// TwinCAT 3 PLC project PLC
// ProgramVersion: 3.1.4024.0
// libraries:
//   Tc2_Standard, * (Beckhoff Automation GmbH)
//   Tc2_System, * (Beckhoff Automation GmbH)
//   Tc3_EventLogger, * (Beckhoff Automation GmbH)
//   Tc3_Module, * (Beckhoff Automation GmbH)
// project tree:
//   GVLs/ GVL.TcGVL
//   / PlcTask.TcTTO
//   POUs/ FB_ALARM.TcPOU, FB_ListenerTest.TcPOU, FB_SampleListener.TcPOU, TYP_ALARM_INTERFACE.TcDUT, MAIN.TcPOU
// real-time tasks:
//   TASK PlcTask: cycle T#10ms, priority 20, ADS port 350

CONFIGURATION PLC
    RESOURCE PLC ON TwinCAT3
        TASK PlcTask(INTERVAL := T#10ms, PRIORITY := 20);
        PROGRAM MAIN WITH PlcTask : MAIN;
    END_RESOURCE
END_CONFIGURATION

// ---- POUs/TYP_ALARM_INTERFACE.TcDUT
TYPE TYP_ALARM_INTERFACE :
STRUCT
	bActivate : BOOL;
	bConfirm : BOOL;
	sMessage : STRING;
	sSourceMessage : STRING;
	nEventID : UDINT;
	nSourceID : UDINT;
END_STRUCT
END_TYPE

// ---- GVLs/GVL.TcGVL
{attribute 'qualified_only'}
VAR_GLOBAL
	{attribute 'OPC.UA.DA' := '1'}
	{attribute 'OPC.UA.DA.StructuredType' := '1'}
	arrAlarms : ARRAY[0..99] OF TYP_ALARMS;
END_VAR

// ---- POUs/MAIN.TcPOU
PROGRAM MAIN
VAR
	GeneralAlarms : ARRAY[0..2] OF TYP_ALARM_INTERFACE :=
	[(nEventID:=3, nSourceID:=101, sMessage:='MESSAGE 1', sSourceMessage:='SOURCE 1'),
	(nEventID:=3, nSourceID:=202, sMessage:='MESSAGE 2', sSourceMessage:='SOURCE 2'),
	(nEventID:=3, nSourceID:=303, sMessage:='MESSAGE 3', sSourceMessage:='SOURCE 3')];
	
	fbGeneralAlarms : ARRAY [0..2] OF FB_ALARM;
	fbListener : FB_ListenerTest;
	bResetArray : BOOL;
	i: INT;
END_VAR

fbListener(arrAlarms:=GVL.arrAlarms);

FOR i:=0 TO 2 BY 1 DO
	fbGeneralAlarms[i](eventEntry:=TC_EVENTS.AlarmEventClass.General_alarm, 
			bEvt := GeneralAlarms[i].bActivate, 
			bConfirm := GeneralAlarms[i].bConfirm,
			sMessage := GeneralAlarms[i].sMessage,
			nUserEventID := GeneralAlarms[i].nEventID,
			nUserSourceID := GeneralAlarms[i].nSourceID,
			sSourceMessage := GeneralAlarms[i].sSourceMessage,
			arrAlarms := GVL.arrAlarms);
END_FOR	
		
IF bResetArray THEN
	memset(ADR(GVL.arrAlarms),0,SIZEOF(GVL.arrAlarms));
	bResetArray := FALSE;
END_IF

END_PROGRAM

// ---- POUs/FB_ALARM.TcPOU
FUNCTION_BLOCK FB_ALARM EXTENDS FB_TcAlarm
VAR_INPUT
	eventEntry : TcEventEntry;
	bEvt : BOOL;
	bConfirm : BOOL;
	nUserEventID : UDINT;
	nUserSourceID : UDINT;
	sMessage : STRING;
	sSourceMessage : STRING;
END_VAR
VAR_IN_OUT
	arrAlarms : ARRAY[*] OF TYP_ALARMS;
END_VAR
VAR_OUTPUT
END_VAR
VAR
	bInit : BOOL := TRUE;
	bMem : BOOL;
	fbMsg : FB_TcMessage;
	fbSourceInformation : FB_TcSourceInfo;
END_VAR

//INITIALISING THE ALARM WHEN THE RAISING OF THE ALARM IS REQUESTED
IF bEvt AND NOT bMem (*AND SUPER^.eConfirmationState <> TcEventConfirmationState.WaitForConfirmation*) THEN
	IF bInit THEN
		fbSourceInformation.Clear();
		fbSourceInformation.sName := sSourceMessage;
		fbSourceInformation.nId := nUserSourceID;
		eventEntry.nEventId := nUserEventID;
		SUPER^.CreateEx(eventEntry, TRUE, ipSourceInfo := fbSourceInformation);
		SUPER^.ipArguments.Clear().AddString(sMessage);
		bInit := FALSE;
	END_IF
END_IF

//AFTER INITIALISING, RAISE THE ALARM
IF NOT bInit THEN
	SUPER^.Raise(0);
	bInit := TRUE;
END_IF

//CLEARING THE ALARM
IF bMem AND NOT bEvt THEN
	SUPER^.Clear(0, FALSE);	
END_IF

//CONFIRMING THE ALARM
IF bConfirm THEN
	SUPER^.Confirm(0);
END_IF

bMem := bEvt;

END_FUNCTION_BLOCK

// ---- POUs/FB_ListenerTest.TcPOU
FUNCTION_BLOCK FB_ListenerTest
VAR_INPUT
END_VAR
VAR_IN_OUT
	arrAlarms : ARRAY[*] OF TYP_ALARMS;
END_VAR
VAR_OUTPUT
END_VAR
VAR
	hr : HRESULT;
	
	bSubscribe : BOOL := TRUE;
	bSubscribed : BOOL;
	bUnSubscribe : BOOL;
	
	fbListenerFilter : FB_TcEventFilter; 
	fbMessageListener : FB_SampleListener;
	
END_VAR

fbMessageListener.arrAlarms := arrAlarms;
fbMessageListener.Execute(); // retrieve messages and its texts

IF bSubscribe THEN 
	bSubscribe := FALSE;
	fbListenerFilter.Clear().EventClass.EqualTo(TC_EVENTS.AlarmEventClass.General_alarm.uuidEventClass); //define all events (messages and alarms) from this eventclass   
	hr := fbMessageListener.Subscribe2(fbListenerFilter); //subscribe to retrieve defined events
	IF SUCCEEDED(hr) THEN	
		bSubscribed := TRUE;
	END_IF
END_IF 

IF bUnSubscribe THEN 
	bUnSubscribe := FALSE;
	hr := fbMessageListener.Unsubscribe();
	IF SUCCEEDED(hr) THEN	
		bSubscribed := FALSE;
	END_IF
END_IF

END_FUNCTION_BLOCK

// ---- POUs/FB_SampleListener.TcPOU
FUNCTION_BLOCK FB_SampleListener EXTENDS FB_ListenerBase2
VAR_INPUT
END_VAR
VAR_IN_OUT
	arrAlarms : ARRAY[*] OF TYP_ALARMS;
END_VAR
VAR_OUTPUT
END_VAR
VAR
	sJsonAttribute : STRING (10000);	
	hr : HRESULT;
	
	nCntMessagesSent : INT;
	nCntAlarmsRaised : INT;
	nCntAlarmsConfirmed : INT;
	nCntAlarmsCleared : INT;
	
	//text retrieval of message
	fbRequestEventText : FB_RequestEventText;
	{attribute 'TcEncoding':='UTF-8'}
	sLastMessageText : STRING;
	bReqText : BOOL;
END_VAR

METHOD Execute : HRESULT
VAR_INPUT
END_VAR
Execute := SUPER^.Execute(); //retrieve events

//retrieve the text of a message
IF 	bReqText AND fbRequestEventText.bError THEN 
	sLastMessageText := 'Error';
	bReqText := FALSE; 
ELSIF bReqText AND NOT  fbRequestEventText.bBusy THEN
	fbRequestEventText.GetString(sLastMessageText, SIZEOF(sLastMessageText));
	bReqText := FALSE;
END_IF
END_METHOD

METHOD OnAlarmCleared : HRESULT
VAR_INPUT
	fbEvent : REFERENCE TO FB_TcEvent;
END_VAR
VAR
	i : INT;
	j : INT;
END_VAR
nCntAlarmsCleared := nCntAlarmsCleared + 1;

FOR i:=0 TO 99 BY 1 DO
	//CYCLING THRU THE ARRAY TO FIND IF A MATCHING ALARM EXISTS
	IF arrAlarms[i].AlarmID = fbEvent.nEventId AND arrAlarms[i].SourceID = fbEvent.ipSourceInfo.nId THEN
		//UPDATING THE CONFIRMED STATE
		arrAlarms[i].isActive := FALSE;	
	END_IF	 
	//IF ALARM IS (CONFIRMED AND NOT ACTIVE) THEN REMOVING THE ALARM FROM THE ARRAY
	IF arrAlarms[i].isConfirmed AND NOT arrAlarms[i].isActive THEN
		FOR j:=i TO 99 BY 1 DO
			arrAlarms[j]:=arrAlarms[j+1];
		END_FOR
	END_IF	
END_FOR

OnAlarmCleared := S_OK; // in order to receive more callbacks (Set <> S_OK in order to cancel the callbacks for this program cycle.)
END_METHOD

METHOD OnAlarmConfirmed : HRESULT
VAR_INPUT
	fbEvent : REFERENCE TO FB_TcEvent;
END_VAR
VAR
	i : INT;
	j: INT;
END_VAR
nCntAlarmsConfirmed := nCntAlarmsConfirmed + 1;

FOR i:=0 TO 99 BY 1 DO
	//CYCLING THRU THE ARRAY TO FIND IF A MATCHING ALARM EXISTS
	IF arrAlarms[i].AlarmID = fbEvent.nEventId AND arrAlarms[i].SourceID = fbEvent.ipSourceInfo.nId THEN
		//UPDATING THE CONFIRMED STATE
		arrAlarms[i].isConfirmed := TRUE;	
	END_IF	
	//IF ALARM IS (CONFIRMED AND NOT ACTIVE) THEN REMOVING THE ALARM FROM THE ARRAY
	IF arrAlarms[i].isConfirmed AND NOT arrAlarms[i].isActive THEN
		FOR j:=i TO 99 BY 1 DO
			arrAlarms[j]:=arrAlarms[j+1];
		END_FOR
	END_IF	 
END_FOR

OnAlarmConfirmed := S_OK; // in order to receive more callbacks (Set <> S_OK in order to cancel the callbacks for this program cycle.)
END_METHOD

METHOD OnAlarmRaised : HRESULT
VAR_INPUT
	fbEvent : REFERENCE TO FB_TcEvent;
END_VAR
VAR
	i : INT;
END_VAR
hr := fbEvent.GetJsonAttribute(sJsonAttribute, SIZEOF(sJsonAttribute));
nCntAlarmsRaised := nCntAlarmsRaised + 1;

//MOVING ALL ALARM ARRAY MEMBERS BACK BY 1
FOR i:=99 TO 1 BY -1 DO
		arrAlarms[i]:=arrAlarms[i-1];
END_FOR
//ENTERING THE NEW ALARM TO THE FIRST PLACE OF THE ARRAY
arrAlarms[0].AlarmID:=fbEvent.nEventId;
arrAlarms[0].SourceID:=fbEvent.ipSourceInfo.nId;
arrAlarms[0].SourceName:=fbEvent.ipSourceInfo.sName;
arrAlarms[0].isActive := TRUE;
arrAlarms[0].isConfirmed := FALSE;

OnAlarmRaised := S_OK; // in order to receive more callbacks (Set <> S_OK in order to cancel the callbacks for this program cycle.)
END_METHOD

METHOD OnMessageSent : HRESULT
VAR_INPUT
	fbEvent : REFERENCE TO FB_TcEvent;
END_VAR

VAR 
END_VAR
hr := fbEvent.GetJsonAttribute(sJsonAttribute, SIZEOF(sJsonAttribute));
nCntMessagesSent := nCntMessagesSent + 1;

fbRequestEventText.Request(eventClass:=fbEvent.EventClass, nEventId:=fbEvent.nEventId, nLangId:=1033, ipArgs:=fbEvent.ipArguments );
bReqText := TRUE;

OnMessageSent := S_OK; // in order to receive more callbacks (Set <> S_OK in order to cancel the callbacks for this program cycle.)
END_METHOD

END_FUNCTION_BLOCK
